TEXTLIST TL_MessageDiscriptions
  0 = 'No message active'
  1 = 'Unknown error occured'
  2 = 'No communication detected'
  3 = 'Communication error detected (does not match expected com)'
  4 = 'Hardware overload detected'
  5 = 'Encoder signal incorrect or not present'
  6 = 'Slave system is has active fatal fault'
  7 = 'Axis fault feedback'
  8 = 'Axis drive fault'
  9 = 'Collision detected between 2 or more parts of the machine'
  100 = 'Hardware feedback is does not match expected'
  101 = 'Hardware moving in incorrect direction'
  102 = 'Hardware movement completion time is lower then minimum'
  103 = 'Hardware movement maximum time was exceeded'
  104 = 'Hardware is at different position then expected'
  105 = 'Obstruction detected in movement path'
  200 = 'Waiting for product'
  201 = 'Waiting for operator action'
  202 = 'Waiting for other module'
  203 = 'Waiting Waiting for master'
  204 = 'Waiting for slave'
  205 = 'Action or command not possible in current position'
  300 = 'Product is almost empty refif is required'
  301 = 'Product or action is finished'
  302 = 'Ready for new task'
  900 = 'Fatal fault message test'
  901 = 'Cycle fault message test'
  902 = 'Missing condition message test'
  903 = 'Operator message test'
   = ''
END_TEXTLIST

(* stored: Version 1.1.0.1, ProductVersion 3.1.4024.3
   TextList TL_MessageDiscriptions: Id {0743355f-7906-4af3-9248-c2492f12cce9} *)
